FUNCTION TFGetNearestWA : ARRAY [1..MAXAREA] OF TFMachinePalletizer_WorkAreaSort
VAR_INPUT
	WorkArea : POINTER TO ARRAY [1..MAXAREA] OF TFMachinePalletizer_WorkArea;
	WorkPickPoint : TFMachinePalletizer_WorkPickPointSlab;
END_VAR
VAR
	DistanceFromWA : ARRAY [1..MAXAREA] OF TFMachinePalletizer_WorkAreaSort;
	WAS : TFMachinePalletizer_WorkAreaSort;
	i : INT;
	j : INT;
	k : INT;
	c : INT;
END_VAR


FOR i:=1 TO MAXAREA DO
	DistanceFromWA[i].Distance:= 0;
	DistanceFromWA[i].cwa:= 0;
END_FOR

FOR j:=1 TO MAXAREA DO
	IF WorkArea^[j].X > 0 THEN
		DistanceFromWA[j].Distance := ABS(WorkPickPoint.X - WorkArea^[j].X); 
		DistanceFromWA[j].cwa := j;
	END_IF
END_FOR

(* Bubble Sort *)
FOR k:=1 TO MAXAREA DO
	FOR c:=1 TO MAXAREA DO
		IF DistanceFromWA[MAXAREA-c].Distance > DistanceFromWA[MAXAREA-c+1].Distance THEN
			WAS := DistanceFromWA[MAXAREA-c];
			DistanceFromWA[MAXAREA-c] := DistanceFromWA[MAXAREA-c+1];
			DistanceFromWA[MAXAREA-c+1] := WAS;
		END_IF
	END_FOR
END_FOR
TFGetNearestWA := DistanceFromWA;

END_FUNCTION

(* stored: Version 1.1.0.1, ProductVersion 3.1.4024.11
   POU TFGetNearestWA: Id {1a845c6e-bbfc-4348-bd3b-6d3d6b0f2a94}, SpecialFunc None *)
